FUNCTION_BLOCK PNP_CTL_FBD (* Pick and Place AUTO Control with FBD Algorithm *)
  (* Standard: IEC 61499; ApplicationDomain: Discrete Assembly; Function: Pick&Place *)
  (* Version 0.0, 2006-09-18, JHC, Holobloc Inc, Adapted from PNP_CTL_LD. *)
  (* Compiler header: package fb.rt.mach; *)
  (* Compiler classdef: SimpleFB *)
  (* Compiler Java Sun JDK 1.5.0 *)
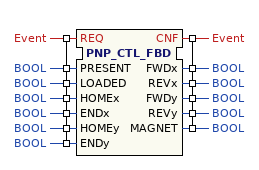
  EVENT_INPUT
    REQ WITH HOMEx, ENDx, HOMEy, ENDy, PRESENT, LOADED; (* Execute control if AUTO mode is ON *)
  END_EVENT
  EVENT_OUTPUT
    CNF WITH FWDx, FWDy, REVy, REVx, MAGNET; (* AUTO mode control executed *)
  END_EVENT
  VAR_INPUT
    PRESENT : BOOL; (* Workpiece Sensor at end of Conveyor *)
    LOADED : BOOL; (* Workpiece Sensor on XY transport *)
    HOMEx : BOOL; (* x-axis at HOME position *)
    ENDx : BOOL; (* x-axis at END position *)
    HOMEy : BOOL; (* y-axis at HOME position *)
    ENDy : BOOL; (* y-axis at END position *)
  END_VAR
  VAR_OUTPUT
    FWDx : BOOL; (* Drive x-axis Motor Forward (toward ENDx) *)
    REVx : BOOL; (* Drive x-axis Motor 1 in Reverse (toward HOMEx) *)
    FWDy : BOOL; (* Drive y-axis Motor Forward (toward ENDy) *)
    REVy : BOOL; (* Drive y-axis Motor 2 in Reverse (toward HOMEy) *)
    MAGNET : BOOL; (* Electromagnet ON (grasp workpiece) *)
  END_VAR
  ALGORITHM REQ IN FBD: (* AUTO control algorithm *)
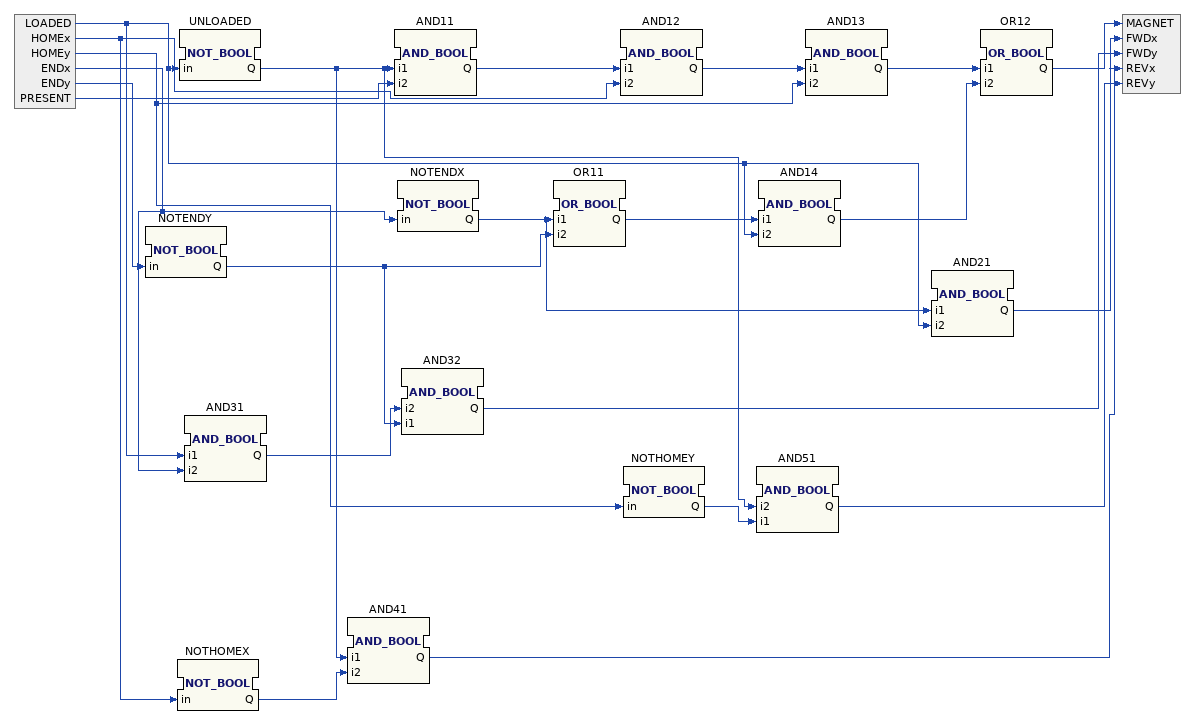
    FBS
      UNLOADED : NOT_BOOL;
      NOTHOMEX : NOT_BOOL;
      NOTHOMEY : NOT_BOOL;
      NOTENDX : NOT_BOOL;
      NOTENDY : NOT_BOOL;
      AND11 : AND_BOOL;
      AND12 : AND_BOOL;
      AND13 : AND_BOOL;
      OR12 : OR_BOOL;
      OR11 : OR_BOOL;
      AND14 : AND_BOOL;
      AND21 : AND_BOOL;
      AND31 : AND_BOOL;
      AND32 : AND_BOOL;
      AND41 : AND_BOOL;
      AND51 : AND_BOOL;
    END_FBS
    DATA_CONNECTIONS
      LOADED TO UNLOADED.in;
      HOMEx TO NOTHOMEX.in;
      HOMEy TO NOTHOMEY.in;
      ENDx TO NOTENDX.in;
      ENDy TO NOTENDY.in;
      UNLOADED.Q TO AND11.i1;
      PRESENT TO AND11.i2;
      AND11.Q TO AND12.i1;
      HOMEx TO AND12.i2;
      AND12.Q TO AND13.i1;
      HOMEy TO AND13.i2;
      AND13.Q TO OR12.i1;
      OR12.Q TO MAGNET;
      NOTENDX.Q TO OR11.i1;
      NOTENDY.Q TO OR11.i2;
      OR11.Q TO AND14.i1;
      LOADED TO AND14.i2;
      AND14.Q TO OR12.i2;
      NOTENDX.Q TO AND21.i1;
      LOADED TO AND21.i2;
      AND21.Q TO FWDx;
      LOADED TO AND31.i1;
      ENDx TO AND31.i2;
      AND31.Q TO AND32.i2;
      NOTENDY.Q TO AND32.i1;
      AND32.Q TO FWDy;
      AND41.Q TO REVx;
      UNLOADED.Q TO AND41.i1;
      NOTHOMEX.Q TO AND41.i2;
      AND51.Q TO REVy;
      UNLOADED.Q TO AND51.i2;
      NOTHOMEY.Q TO AND51.i1;
    END_CONNECTIONS
  END_ALGORITHM
END_FUNCTION_BLOCK
